PROGRAM TEST_MAIN
VAR

cbBlock1 : CommandBlockBase;
cbBlock2 : CommandBlockBase;

cbBlock3 : CommandBlockPos;
cbBlock4 : CommandBlockPos;

ptBlock : POINTER TO CommandBlockBase := ADR(cbBlock1);	
ptBlockPos : POINTER TO CommandBlockPos;

aSize : INT;


memoryPool : ARRAY[1..1024] OF WORD;

ptRunIndexerMaster : POINTER TO RunUnitIndexerMaster;
ptRunGeneric : POINTER TO RunUnitGeneric;

ptUnitGeneric : POINTER TO UnitBase;
ptUnitIndexerMaster : POINTER TO UnitIndexerMaster;

bInitialized : BOOL ;
nCounter : INT ;

simuObstacleSensor : BOOL;
simuReachSensor : BOOL;

tmpObstacleSensorat AT%I*  : BOOL;
tmpReachSensor AT%I* : BOOL;

lifterCelluarA : RunLifterCelluar(argParent:= ADR(lifterCelluarA), 
argSlotBase:= ADR(GVL.MATERIAL_SLOTS[1]), 
argSlotLast:= ADR(GVL.MATERIAL_SLOTS[2]),
argAxis:= ADR(GVL.axisControls[4]),
argCylinder:=ADR(GVL.cylinderControls[1]),
argHit:=ADR(GVL.commandBlocks[16]),
argRelease:=ADR(GVL.commandBlocks[17]),
argWorking:=ADR(GVL.commandBlocks[18]),
argObstacleSensor:= ADR(simuObstacleSensor),
argReachSensor:= ADR(simuReachSensor)
);

masterProxy : RunUnitIndexerMasterCelluarA(argParent:= ADR(masterProxy), 
argSlotBase:= 0, 
argSlotLast:= 0,
argAxis:=0,
argUpstream:=0,
argCommandFast:=0,
argCommandSlow:=0,
argCommandTriggerRaise:=0,
argCommandCheckRaise:=0);

masterCelluarA : RunUnitIndexerMasterCelluarA(argParent:= ADR(masterCelluarA), 
argSlotBase:= ADR(GVL.MATERIAL_SLOTS[1]), 
argSlotLast:= ADR(GVL.MATERIAL_SLOTS[2]),
argAxis:=ADR(GVL.axisControls[1]),
argUpstream:=ADR(masterProxy),
argCommandFast:=ADR(GVL.commandBlocks[32]),
argCommandSlow:=ADR(GVL.commandBlocks[33]),
argCommandTriggerRaise:=ADR(GVL.commandBlocks[40]),
argCommandCheckRaise:=ADR(GVL.commandBlocks[41]));

simuStation : RunUnitGeneric(argParent:= ADR(simuStation), argSlotBase:= ADR(GVL.MATERIAL_SLOTS[1]), argSlotLast:= ADR(GVL.MATERIAL_SLOTS[1]));

END_VAR

cbBlock1.AXIS_ID:=5;
ptBlock:=ADR(cbBlock1);

cbBlock2:=ptBlock^; // value assignment?
//change cbBlock1 , watch if cbBlock2 changed

ptBlock := ADR(cbBlock3); //if possible mophism

cbBlock3.COORDINATE:=1234;

ptBlockPos:=ptBlock;
cbBlock4:=ptBlockPos^;//check


//may access violation??
//ptBlockPos:=ADR(cbBlock1);
//ptBlockPos^.COORDINATE:=5555; //may violation

//TEST2();
//TEST_CYLINDER();
//TEST_UNIT_VIRTUAL();
//TEST_UNIT_MASTER();
//TEST_AXIS();
IF NOT bInitialized THEN
	FOR nCounter:=8 TO 64 BY 1 DO
		GVL.commandBlocks[nCounter].command := eCommandTypes.POSITION;
		GVL.commandBlocks[nCounter].parameter.position.Acceleration := 4000;
		GVL.commandBlocks[nCounter].parameter.position.Deceleration := 4000;
		GVL.commandBlocks[nCounter].parameter.position.Velocity := 100;
	END_FOR
	GVL.commandBlocks[8].parameter.position.Position := 300;
	GVL.commandBlocks[8].parameter.position.Velocity := 400;
	
	GVL.commandBlocks[9].parameter.position.Position := 400;
	GVL.commandBlocks[9].parameter.position.Velocity := 100;
	
	GVL.commandBlocks[10].parameter.position.Position := 800;
	GVL.commandBlocks[10].parameter.position.Velocity := 400;
	
	bInitialized := TRUE;
	
	FOR nCounter:=16 TO 18 BY 1 DO
		GVL.commandBlocks[nCounter].parameter.position.Velocity :=35;
		GVL.commandBlocks[nCounter].parameter.position.Acceleration :=1000;
		GVL.commandBlocks[nCounter].parameter.position.Deceleration :=1000;
	END_FOR
	GVL.commandBlocks[16].parameter.position.Position := 4.5;
	GVL.commandBlocks[17].parameter.position.Position := 0;
	GVL.commandBlocks[18].parameter.position.Position := 20;
	//
	GVL.commandBlocks[32].parameter.position.Position :=350;
	GVL.commandBlocks[32].parameter.position.Velocity :=250;
	
	GVL.commandBlocks[33].parameter.position.Position :=410;
	GVL.commandBlocks[33].parameter.position.Velocity :=100;
	
	GVL.commandBlocks[40].parameter.position.Position :=260;
	GVL.commandBlocks[41].parameter.position.Position :=340;
	
	lifterCelluarA.ptObstacleSensorStatus := ADR(tmpObstacleSensorat);
	lifterCelluarA.ptReachSensorStatus := ADR(tmpReachSensor);
END_IF
//TEST_BUFFERING();
//TEST_CYLINDER();

FOR nCounter:=1 TO 8 BY 1 DO
	GVL.axisControls[nCounter]();
	GVL.cylinderControls[nCounter]();
END_FOR

simuStation(
	bEnStep:= , 
	bTrigStep:= , 
	bPause:= , 
	bIsBypassed:= , 
	bWorkingOverride:= , 
	bMaterialOverride:= , 
	State=> , 
	NextState=> , 
	AlarmCode=> );
lifterCelluarA(
	bEnStep:= , 
	bTrigStep:= , 
	bPause:= , 
	bIsBypassed:= , 
	bWorkingOverride:= , 
	bMaterialOverride:= , 
	State=> , 
	NextState=> , 
	AlarmCode=> );
masterCelluarA(
	bEnStep:= , 
	bTrigStep:= , 
	bPause:= , 
	bIsBypassed:= , 
	bWorkingOverride:= , 
	bMaterialOverride:= , 
	State=> , 
	NextState=> , 
	AlarmCode=> , 
	syncAcknowledged:= , 
	slaveLinkageStatus:= , 
	slaveWorkingSignal:= , 
	syncEngaged=> , 
	syncMaterialId=> );
lifterCelluarA.IsHit := masterCelluarA.triggerHit;
lifterCelluarA.IsReleased := masterCelluarA.triggerRelease;
masterCelluarA.allHit := lifterCelluarA.IsHit;
masterCelluarA.allReach := lifterCelluarA.IsReach;
masterCelluarA.allRelease := lifterCelluarA.IsReleased;

//fbCylinder(ptBlock:= ADR(cylinderBlock));

//fbRunIndexerMaster(ptBlock:= );


//no need
//ptRunIndexerMaster := ADR(memoryPool[1]); // fine?
//ptRunGeneric := ADR(memoryPool[1+SIZEOF(ptRunIndexerMaster)]);

//ptRunIndexerMaster^();
//ptRunGeneric^();


//possible manipulate memory allocation
ptUnitGeneric := ADR(memoryPool[1]);
ptUnitIndexerMaster := ADR(memoryPool[1+SIZEOF(ptUnitGeneric^)]);

ptUnitGeneric^.alarmCode := 99;  //

END_PROGRAM

(* stored: Version 1.1.0.1, ProductVersion 3.1.4022.10
   POU TEST_MAIN: Id {c5d24ec2-dcd4-432d-b366-2840b187b342}, SpecialFunc None *)
